(* PLC project Generated.project, CODESYS CODESYS V3.5 SP19 Patch 1 *)
(* stored: creationDateTime 2026-09-06T13:00:42.463208, modificationDateTime 2026-09-06T13:00:42.463208 *)

(* ======================================================================= 🔄 FB_MirrorBypassRetain — Miroir bidirectionnel IHM ↔ RETAIN (bypass) ─────────────────────────────────────────────────────────────── 🎯 Rôle : Synchronise un bypass IHM (volatile) avec sa copie RETAIN (survit à une coupure) — dernier-écrit-gagne : si l'IHM a changé depuis le cycle précédent, le RETAIN suit ; sinon l'IHM est réaligné sur le RETAIN (ex. redémarrage à chaud). 🔌 Architecture : Brique technique sans cycle de vie (pas de défaut à remonter) 📍 Domaine : CODE/J_SUPERVISION (seul consommateur actuel : PRG_07_Supervision §2c) 📄 Doc métier : DOC/STDS/CODE_QUALITY_STANDARDS.md §10 ======================================================================= *)
FUNCTION_BLOCK FB_MirrorBypassRetain
  VAR_IN_OUT
    Hmi : BOOL;  (* === MIROIR BIDIRECTIONNEL === <-> [BUS] Valeur bypass côté IHM (GVL_IHM) *)
    RetainVal : BOOL;  (* <-> [BUS] Valeur bypass côté RETAIN (GVL_PERSISTENT) *)
    Prev : BOOL;  (* <-> [BUS] Mémoire du cycle précédent (détection front IHM) *)
  END_VAR

            

IF Hmi <> Prev THEN
    RetainVal := Hmi;
ELSE
    Hmi := RetainVal;
END_IF;
Prev := Hmi;

          
END_FUNCTION_BLOCK
